FUNCTION_BLOCK FB_ControllerArm EXTENDS FB_StateMachine  IMPLEMENTS I_StateMachine
VAR_INPUT 
	bStartSelftest : BOOL;
	bStartErgonomics : BOOL;
	bStartTeleoperation : BOOL;
	
END_VAR
VAR
	eInnerState : E_ControllerArmStates;

	bDocked : BOOL;

	fbSelfTest : FB_SelfTest;
	fbErgonomics : FB_Ergonomics;
	stErgoCommands : ST_ErgoCommands;
	
	fbStepper : FB_Stepper;
	fbLinearActuator : FB_LinearActuator;
	fbJointSR : FB_Joint;
END_VAR

OuterLopSM();

PROPERTY Calibrated : BOOL
GET
IF bActive THEN
	Calibrated :=  NOT fbSelfTest.SelftestNeeded;
ELSE
	Calibrated := TRUE;	
END_IF
END_GET
END_PROPERTY

METHOD Disable : BOOL

VAR
	bChildBusy: BOOL;
END_VAR
bBusy := TRUE;
fbStepper(bActive:=FALSE);
fbLinearActuator(bActive:=FALSE);
fbJointSR(bActive:=FALSE);
fbSelfTest(bActive:=FALSE);

IF fbStepper.Busy THEN
	bChildBusy := TRUE;
ELSIF fbStepper.bError THEN
	bChildBusy := TRUE;
	//	Stack trace and bError switching are reserved for inner loop
	fbStepper.ErrorAck:=TRUE;
END_IF

IF fbLinearActuator.Busy THEN
	bChildBusy := TRUE;
ELSIF fbLinearActuator.bError THEN
	bChildBusy := TRUE;
	//	Stack trace and bError switching are reserved for inner loop
	fbLinearActuator.ErrorAck:=TRUE;
END_IF

IF fbJointSR.Busy THEN
	bChildBusy := TRUE;
ELSIF fbJointSR.bError THEN
	bChildBusy := TRUE;
	//	Stack trace and bError switching are reserved for inner loop
	fbJointSR.ErrorAck:=TRUE;
END_IF


IF fbSelftest.Busy THEN
	bChildBusy := TRUE;
ELSIF fbSelftest.bError THEN
	bChildBusy := TRUE;
	//	Stack trace and bError switching are reserved for inner loop
	fbSelftest.ErrorAck:=TRUE;
END_IF



IF bChildBusy THEN
	Disable := FALSE;
ELSE
	ChangeInnerState(E_ControllerArmStates.Idle);
	Disable := TRUE;
END_IF
END_METHOD

PROPERTY Docked : BOOL
GET
IF bActive THEN
	Docked := bDocked;
ELSE
	Docked := TRUE;
END_IF
END_GET
END_PROPERTY

PROPERTY ErgoCommands : ST_ErgoCommands
GET
END_GET
SET
{warning 'TODO: update ErgoCommands setter'}
END_SET
END_PROPERTY

PROPERTY Failed : BOOL
GET
Failed := (NOT THIS^.Busy) AND THIS^.bError;
END_GET
END_PROPERTY

METHOD InnerLoopSM : BOOL
VAR_INST
	nI : INT;	
END_VAR
// update all children FBs
fbStepper();
fbLinearActuator();
fbJointSR();
fbSelfTest();

CASE CyclicInnerCase(TO_STRING(eInnerState)) OF
	E_ControllerArmStates.Idle:
		IF bStartSelftest THEN
			bStartSelftest := FALSE;
			ChangeInnerState(E_ControllerArmStates.Selftest1);
		ELSIF bStartErgonomics THEN
			bStartErgonomics := FALSE;
			ChangeInnerState(E_ControllerArmStates.Ergonomics1);
		ELSIF bStartTeleoperation THEN
			bStartTeleoperation := FALSE;
			ChangeInnerState(E_ControllerArmStates.Teleoperation1);
		END_IF
	
	E_ControllerArmStates.Selftest1:
		IF fbSelfTest.Busy THEN
			// fbSelfTest should never be busy here 	
			sErrorDetails := 'fbSelfTest.Busy = TRUE';
			fbEventHandler(eNapID:=E_Event.UNABLE_TO_START_TASK,sMessage:=sErrorDetails);
			bError := TRUE;
		ELSE
			IF fbSelfTest.bError THEN
				sErrorDetails := 'fbSelfTest.bReady=FALSE';
				fbEventHandler(eNapID:=E_Event.UNABLE_TO_START_TASK,sMessage:=sErrorDetails);
				bError := TRUE;
			ELSE
				fbSelfTest.bStart:=TRUE;
				ChangeInnerState(E_ControllerArmStates.Selftest2);
			END_IF
		END_IF

		
	E_ControllerArmStates.Selftest2:
		IF fbSelfTest.Busy THEN
			IF Docked THEN
				// Wait... fbSelftest still active
			ELSE
				sErrorDetails := 'Arm undocked during Self Test';
				fbEventHandler(eNapID:=E_Event.UNDOCKED,sMessage:=sErrorDetails);
				bError := TRUE;
			END_IF
		ELSE
			IF fbSelfTest.bError THEN
				fbEventHandler(eNapID:=E_Event.TASK_FAILED,sTrace:=fbSelfTest.EventTrace);
				fbSelfTest.ErrorAck:=TRUE;
				bError := TRUE;
			ELSE
				IF Calibrated THEN
					fbEventHandler(eNapID:=E_Event.REQUEST_COMPLETED);
					ChangeInnerState(E_ControllerArmStates.Idle);
				ELSE
					sErrorDetails := 'Calibrated=FALSE';
					fbEventHandler(eNapID:=E_Event.TASK_FAILED,sMessage:=sErrorDetails);
					bError := TRUE;
				END_IF
			END_IF
		END_IF
		
	E_ControllerArmStates.Ergonomics1:
		IF fbErgonomics.Busy THEN
			// Wait... fbErgonomics still active
		ELSE
			IF fbErgonomics.bError THEN
				fbEventHandler(eNapID:=E_Event.UNABLE_TO_START_TASK,sTrace:=fbErgonomics.EventTrace);
				fbErgonomics.ErrorAck:=TRUE;
				bError := TRUE;
			ELSE
				fbErgonomics.bStart := TRUE;
				ChangeInnerState(E_ControllerArmStates.Ergonomics2);
			END_IF
		END_IF
		
	E_ControllerArmStates.Ergonomics2:
		IF fbErgonomics.Busy THEN
			IF fbErgonomics.Waiting THEN
				// fbErgonomics ready for new command
				fbErgonomics.ErgoCommands := stErgoCommands;
			ELSE
				// Wait... fbErgonomics is still performing a task
			END_IF
		ELSE
			IF fbErgonomics.bError THEN
				fbEventHandler(eNapID:=E_Event.TASK_FAILED,sTrace:=fbErgonomics.EventTrace);
				fbErgonomics.ErrorAck:=TRUE;
				bError := TRUE;
			ELSE
				ChangeInnerState(E_ControllerArmStates.Idle);
			END_IF
		END_IF
	
		E_ControllerArmStates.Teleoperation1:
			// TODO
		
			

END_CASE
END_METHOD

METHOD PUBLIC ReadStatus : BOOL
fbStepper.ReadStatus();
{warning 'TODO: add all hardware children to ControllerArm.ReadStatus()'}
END_METHOD

PROPERTY Ready : BOOL
GET
Ready := (NOT THIS^.Busy) AND (NOT bError);
END_GET
END_PROPERTY

METHOD Reset : BOOL
// reset variables specific to this FB 
bStartSelftest := FALSE;
bStartErgonomics := FALSE;
bStartTeleoperation := FALSE;

// Reactivate children FBs
fbSelfTest.Active:=TRUE;
fbStepper.Active:=TRUE;
fbLinearActuator.Active:=TRUE;
fbJointSR.Active:=true;
END_METHOD

METHOD Setup : BOOL
eStateMachineSourceID := eStateSourceID;

fbStepper(eStateSourceID := THIS^.eStateMachineSourceID +  E_ArmID_Offset.StepperMotor,
					aErrorLog:=THIS^.aErrorLog,
					nErrorLogIndex:=THIS^.nErrorLogIndex);
					
fbLinearActuator(eStateSourceID := THIS^.eStateMachineSourceID +  E_ArmID_Offset.LinearActuator,
					aErrorLog:=THIS^.aErrorLog,
					nErrorLogIndex:=THIS^.nErrorLogIndex);

fbJointSR(eStateSourceID := THIS^.eStateMachineSourceID +  E_ArmID_Offset.ShoulderRollJoint,
					aErrorLog:=THIS^.aErrorLog,
					nErrorLogIndex:=THIS^.nErrorLogIndex);

fbSelfTest(eStateSourceID := THIS^.eStateMachineSourceID +  E_ArmID_Offset.SelfTest,
					aErrorLog:=THIS^.aErrorLog,
					nErrorLogIndex:=THIS^.nErrorLogIndex,
					fbStepper:=THIS^.fbStepper,
					fbLinearActuator:=THIS^.fbLinearActuator,
					fbJointSR:=THIS^.fbJointSR);
					
fbErgonomics(eStateSourceID := THIS^.eStateMachineSourceID +  E_ArmID_Offset.SelfTest,
					aErrorLog:=THIS^.aErrorLog,
					nErrorLogIndex:=THIS^.nErrorLogIndex,
					fbStepper:=THIS^.fbStepper,
					fbLinearActuator:=THIS^.fbLinearActuator);
					
SetInnerEnumeration(nStateEnum:=THIS^.eInnerState);
END_METHOD

PROPERTY StartErgonomics : BOOL
GET
StartErgonomics := bStartErgonomics;
END_GET
SET
bStartErgonomics := StartErgonomics;
END_SET
END_PROPERTY

PROPERTY StartSelftest : BOOL
GET
StartSelftest := bStartSelftest;
END_GET
SET
bStartSelftest := StartSelftest;
END_SET
END_PROPERTY

PROPERTY StartTeleoperation : BOOL
GET
StartTeleoperation:=bStartTeleoperation;
END_GET
SET
bStartTeleoperation := StartTeleoperation;
END_SET
END_PROPERTY

PROPERTY StopMotors : BOOL
GET
END_GET
SET
END_SET
END_PROPERTY

END_FUNCTION_BLOCK

(* stored: Version 1.1.0.1, ProductVersion 3.1.4024.12
   POU FB_ControllerArm: Id {9d97f625-9b2c-4231-b0c1-617fba0df57d}, SpecialFunc None
   Folder Properties: Id {131f4f8b-9880-4af5-9615-5ef2ac06ece9}
   Property Calibrated: Id {49ba6a80-5e5e-43a5-8db5-e7121236d63d}
   Get Get: Id {8757163b-35a7-4755-8bf0-0f1788bf32d3}
   Method Disable: Id {c2eeebb9-16fe-41d5-8a9c-f26afa1abbd2}
   Property Docked: Id {bc3dbaaa-ebd0-413f-99ac-717967aac553}
   Get Get: Id {2cea9a5c-f783-42cb-84d9-50319bdc5492}
   Property ErgoCommands: Id {52474e6d-bffd-4a10-b67d-9dfe75d2c671}
   Get Get: Id {2585786c-d097-40f3-877d-89f18bb0d849}
   Set Set: Id {1852afb1-1c53-4151-8729-bcf2204142f6}
   Property Failed: Id {cb0fb621-9372-468b-b0b1-4f3930fbd69a}
   Get Get: Id {da5b53b5-7d72-444f-8771-6cdefc5b07eb}
   Method InnerLoopSM: Id {7047a9cc-bc34-4004-85b2-a2bd1ace4e67}
   Method ReadStatus: Id {d0017fc7-2b4c-43b5-a68e-d6f255f1e562}
   Property Ready: Id {02b0be2d-fbe2-48a8-b559-8b4c768564ff}
   Get Get: Id {a6ad0bf9-3778-407c-b19f-3ca60c2d84fb}
   Method Reset: Id {d744f583-81d0-40a6-a3fe-9e7e7aae722f}
   Method Setup: Id {2a86b95f-c957-4ac0-903c-e7b6b06c7117}
   Property StartErgonomics: Id {7b4dc2a8-5723-4fbb-bcf0-54feacd33e46}
   Get Get: Id {c322d885-c869-4fef-b1ad-9883f4df29f8}
   Set Set: Id {46122d6a-544e-427f-8fe1-f6da4f65fa58}
   Property StartSelftest: Id {25f59324-1551-45f5-8872-bcf4c5541c6b}
   Get Get: Id {78c6e660-984c-4093-83ab-c67284c3e1fa}
   Set Set: Id {f016e3dc-c0e5-4821-9579-d3b1f254da1b}
   Property StartTeleoperation: Id {bf51e4c0-aa20-4fdb-9e1a-a7a66633bbd8}
   Get Get: Id {2093e615-d01c-4135-8bf2-16240e850889}
   Set Set: Id {9cb997d5-87e4-4832-a647-4d7a1024b427}
   Property StopMotors: Id {9529c5fc-0525-4349-92c6-149c11bd727d}
   Get Get: Id {e4a6c671-58ae-41d7-81e5-e3678cb9e2e6}
   Set Set: Id {10029bb0-a4bf-4751-9087-bbe2b960a97b} *)
